{attribute 'linkalways'} 
{attribute 'no_explicit_call' := 'This FB is a CLASS and must be accessed using methods or properties'}
{attribute 'enable_dynamic_creation'}
FUNCTION_BLOCK Node_F_VN_GetAt_REAL EXTENDS VisionNode
VAR
    ipContainer : _ITcVnContainer;
    fElement : _REAL(0);
    nIndex : _ULINT(0);
    hrPrev : _HRESULT(S_OK);
    hresult : _HRESULT(S_OK);
END_VAR

METHOD PUBLIC  Clone : I_Node
VAR
	pNode : POINTER TO Node_F_VN_GetAt_REAL;
END_VAR
pNode := __NEW(Node_F_VN_GetAt_REAL);
Clone := pNode^;
END_METHOD

METHOD FB_init : BOOL
VAR_INPUT
	bInitRetains : BOOL; // if TRUE, the retain variables are initialized (warm start / cold start)
	bInCopyCode : BOOL;  // if TRUE, the instance afterwards gets moved into the copy code (online change)
END_VAR
AddInput('ipContainer', ipContainer);
AddParameter('nIndex', nIndex);
AddInput('hrPrev', hrPrev);
AddOutput('fElement', fElement);
AddOutput('hresult',hresult);
END_METHOD

METHOD PROTECTED OnExecute
hresult.Value := F_VN_GetAt_REAL(
    ipContainer := ipContainer.Value,
    fElement := fElement.Value,
    nIndex := nIndex.Value,
    hrPrev:= hrPrev.Value);
END_METHOD

METHOD PUBLIC PreExecutionCheck
VAR_INPUT
	Check : I_PreExecutionChecks;
END_VAR
Check.IsTrue(ipContainer.IsValid, 'ipContainer must be a valid container');
Check.IsTrue(ipContainer.IsType(TC_GLOBAL_CONST_LIST.ContainerType_Vector_REAL), 'ipContainer contains incorrect type');
END_METHOD

END_FUNCTION_BLOCK

(* stored: Version 1.1.0.1, ProductVersion 3.1.4026.13
   POU Node_F_VN_GetAt_REAL: Id {3e76de2c-1b8c-40ff-a514-9010fd6c8296}, SpecialFunc None
   Folder Constructor: Id {8dcb89de-1b5a-40b6-9ec6-59864ae05a74}
   Method Clone: Id {19d52e04-8d13-4a9c-b294-bea1a02bf2a5}
   Method FB_init: Id {d564ae58-c02f-46ca-8b17-b6bd40f4b7bc}
   Method OnExecute: Id {9f96a7a2-c554-4d4d-8582-99c83d8d4b21}
   Method PreExecutionCheck: Id {07279c5c-4cf2-4827-8332-ba37ec805802} *)
